Xinje XCPPro project, PLC1: XC3-32 (software 3.3q)

PROGRAM Ladder

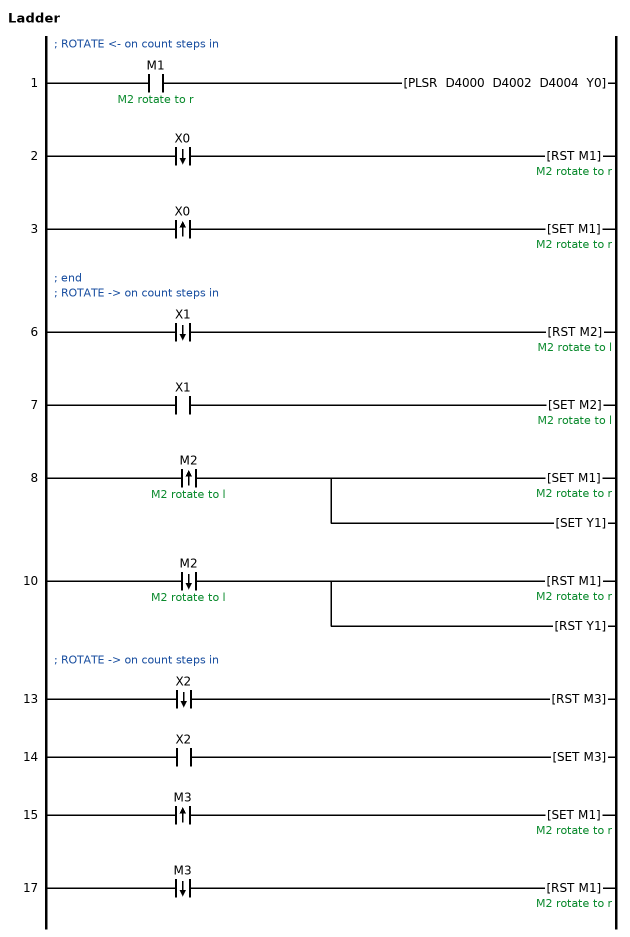
; ROTATE <- on count steps in 
LD     M1	; M2 rotate to r
PLSR   D4000 D4002 D4004 Y0
LDF    X0
RST    M1	; M2 rotate to r
LDP    X0
SET    M1	; M2 rotate to r
; end
; ROTATE -> on count steps in 
LDF    X1
RST    M2	; M2 rotate to l
LD     X1
SET    M2	; M2 rotate to l
LDP    M2	; M2 rotate to l
SET    M1	; M2 rotate to r
SET    Y1
LDF    M2	; M2 rotate to l
RST    M1	; M2 rotate to r
RST    Y1
; ROTATE -> on count steps in 
LDF    X2
RST    M3
LD     X2
SET    M3
LDP    M3
SET    M1	; M2 rotate to r
LDF    M3
RST    M1	; M2 rotate to r